// TIA Portal V17 export
// export: Created 2026-04-13T11:12:44.3951378Z, ExportSetting WithDefaults, DisplayName Totally Integrated Automation Portal, DisplayVersion V17 Update 4, DisplayName TIA Portal Openness, DisplayVersion V17 Update 4, DisplayName TIA Portal Version Control Interface, DisplayVersion V17, DisplayName SINAMICS Startdrive Advanced, DisplayVersion V17, DisplayName SINAMICS Startdrive G130, G150, S120, S150, SINAMICS MV, S210, DisplayVersion V17, DisplayName SINAMICS Startdrive G110M, G120, G120C, G120D, G120P, G115D, DisplayVersion V17, DisplayName STEP 7 Professional, DisplayVersion V17 Update 4, DisplayName STEP 7 Safety, DisplayVersion V17, DisplayName WinCC Professional, DisplayVersion V17 Update 4
DATA_BLOCK "A7-温度控制_DB"   // DB13
VERSION : 0.1
// stored: AutoNumber true, DBAccessibleFromOPCUA true, DBAccessibleFromWebserver true, InstanceOfName A7-温度控制, InstanceOfType FB
"A7-温度控制"
   // VAR
   //    Modbus_Comm_Load { S7_SetPoint := 'True'} : Modbus_Comm_Load;
   //    MB_MASTER { S7_SetPoint := 'True'} : Modbus_Master;
   //    FB_DTC1 { S7_SetPoint := 'True'} : "A1-台达DTC";
   //    FB_DTC2 { S7_SetPoint := 'True'} : "A1-台达DTC";
   //    FB_DTC3 { S7_SetPoint := 'True'} : "A1-台达DTC";
   //    FB_DTC4 { S7_SetPoint := 'True'} : "A1-台达DTC";
   //    FB_DTC5 { S7_SetPoint := 'True'} : "A1-台达DTC";
   //    P { S7_SetPoint := 'True'} : Array[1..16] of Bool;
   //    R_TRIG1 : R_TRIG;
   //    FB_DTC_Instance { S7_SetPoint := 'True'} : "A1-台达DTC";
   //    FB_DTC_Instance_1 { S7_SetPoint := 'True'} : "A1-台达DTC";
   //    通信异常计数 : Array[0..16] of Int;
   //    通信故障 : Array[0..16] of Bool;
   //    总通信故障 : Bool;
   //    i : UDInt;
   // END_VAR
BEGIN
END_DATA_BLOCK
